TYPE ST_ControllerInputs :
STRUCT
	MeassuredValue	: INT;
	ValvePosition	: UINT;
	StatusWord		: UINT;
	AmsAddr			: Tc2_System.ST_AmsAddr;
END_STRUCT
END_TYPE

(* stored: Version 1.1.0.1
   DUT ST_ControllerInputs: Id {2a37d0cc-0bc4-015f-2e64-184cf6af0532} *)
